Universal Robots URScript: SUB_104.script

def SUB_104():
  global _hidden_verificationVariable=0
  set_target_payload(0.100000, [0.135000, 0.000000, 0.225000], [10.000000, 10.000000, 10.000000, 0.000000, 0.000000, 0.000000])
  set_tool_communication(False, 115200, 0, 1, 1.5, 3.5)
  set_tool_output_mode(0)
  set_tool_digital_output_mode(0, 1)
  set_tool_digital_output_mode(1, 1)
  set_tool_voltage(0)
  set_gravity([0.0, 0.0, 9.82])
  set_tcp(p[0.0,0.06,0.535,0.0,0.0,0.0])
  set_safety_mode_transition_hardness(1)
  set_standard_analog_input_domain(0, 1)
  set_standard_analog_input_domain(1, 1)
  set_tool_analog_input_domain(0, 1)
  set_tool_analog_input_domain(1, 1)
  set_analog_outputdomain(0, 0)
  set_analog_outputdomain(1, 0)
  set_input_actions_to_default()
  set_runstate_gp_boolean_output_to_value(0, 3)
  global isReCapt=False
  global Bucket_Z=[0, 0.7]
  global DistPillar=475
  global CandCnt=0
  global lr=1
  global ReCaptZ=0.05
  global forceval=p[0, 0, 0, 0, 0, 0]
  global CaptDepth=[0.24, 0.48]
  global port=3000
  global isOnlyF=True
  global retX2=p[-0.84412, -0.4876, 0.2794, 0, 0, 1.60139]
  global socket_timeout=120
  global isSkipP=False
  global curpos=p[0, 0, 0, 0, 0, 0]
  global host="192.168.2.2"
  global is_popup=False
  global CaptZOffset=0
  global isGoHome=True
  global i_pos2=p[-0.73382, -0.14132, 0.15275, 1.98953, 2, 0.39506]
  global i_pos1=p[-0.73374, -0.14131, 0.15302, 1.98952, 2.00006, 0.39504]
  global pBucket=[p[0.82565, 0.40576, 0.29486, 0, 0, -1.55844], p[-0.84412, -0.4876, 0.2794, 0, 0, 1.60139]]
  global CaptStepZ=0.08
  global CaptIndex=[0, 0]
  global CaptStepX=0.432
  global pBucketM=p[-0.80141, -0.42542, 0.2879, 0, 0, 1.55713]
  global socket_name="vt"
  global rovi_err=0
  global SubPrgResult=800
  global CurrPos=p[-0.54788, -0.05903, 0.40596, -2.14575, -2.29173, -0.02163]
  global CurrPos_p=p[-0.48377, -0.04896, -0.12847, -2.14575, -2.29173, -0.02163]
  global ForceStartZ=9999
  global Bucket=p[0.32604,0.49174,0.0,-1.882900624652718E-5,2.8304179127934987E-5,-1.593185305749222]
  global BucketM=p[0.32604,0.49174,0.0,1.2814539732933814E-16,-2.611297964559462E-16,-1.5931853071795858]
  global CaptPoint_C=p[-0.4219337985373468,-0.003168602281063755,0.36,-2.1962364319980803,-2.243931608455561,-0.021848848268139726]
  global CaptPoint_C2=p[0.32796661698047924,-0.010768520544682924,0.01931625281283378,2.2288103429550152,-2.213636886217198,8.598462540813273E-5]
  global CaptPoint_L1=p[-0.42193494849366175,-0.2,0.36,-2.1962086037526616,-2.243896582262281,-0.02199725151102503]
  global CaptPoint_L2=p[0.327894307417917,-0.010799940826224014,0.01928712668893995,2.087717047309385,-2.0736781215133306,0.27365839887453103]
  global CaptPoint_R1=p[-0.4219551896101372,0.3,0.36,-2.1960823751566156,-2.243954123514977,-0.021863042557794844]
  global CaptPoint_R2=p[0.327926308680866,-0.010795166414457658,0.019300245403843563,-2.1186306375223185,2.1040550557443427,0.22023197678473694]
  global Capt_1BK_L=p[-0.4574214308482636,-0.48457071473611046,0.3504487959434708,-2.1962343446504526,-2.243967222238911,-0.021809195357489434]
  global Capt_1BK_L_kari=p[-0.9062780457975316,-0.3948152887685301,0.3041579389647211,-1.973454285761923,-1.9354309814821136,0.46582663599327684]
  global Capt_1BK_R=p[-0.4574597285646511,0.4755214243904677,0.35039311859649847,-2.196330286580149,-2.2438949166739053,-0.021738621025254933]
  global Capt_1BK_R_kari=p[-0.9062432457725078,0.5951337546911526,0.30410336812750105,-1.9735777661712788,-1.9353884348839347,0.46584435471052615]
  global Capt_1BK_pos1=p[-0.4218793038724447,-0.003154429464978058,0.2915499891144615,-2.1963422029204875,-2.2438663520270015,-0.02197160668673838]
  global Capt_1BK_pos2=p[-0.42187829024618434,-0.0031710253373066375,0.29156503858953065,-2.196324918349679,-2.2439040699490773,-0.021928444416953782]
  global Capt_1BK_pos2_k=p[-0.6125678682784722,-0.030388805985305904,0.07817890571333086,-1.7892541925095446,-1.8765982468297469,0.6168577595976025]
  global Capt_2BK_L=p[0.42186661528427194,0.4254738068040517,0.35042275762909847,2.239156309475874,-2.1837044610999294,0.002643817066643282]
  global Capt_2BK_L_kari=p[1.0654977997166857,0.48819520122022786,0.0997150581225536,-1.8581624430714432,1.7479280549699192,-0.330138866280949]
  global Capt_2BK_R=p[0.4218208572756906,-0.5427676723257963,0.350372239919558,2.2392697861179327,-2.183553596194912,0.002410470905346486]
  global Capt_2BK_R_kari=p[1.0635189639466671,-0.5406292885234477,0.09156512141204048,-2.1417082668537115,1.7859902718169367,-0.7309097134650204]
  global Capt_2BK_pos1=p[0.42193501458435656,0.004742683868356356,0.35045865974037793,2.2391012408536453,-2.1839704655717003,0.002677867056024068]
  global Capt_2BK_pos2=p[0.421903984494575,0.004707988774967922,0.35045218900915065,2.239114367170047,-2.183895515396197,0.002684056681074047]
  global Capt_2BK_pos2_k=p[0.4977433025854323,-0.009744988529796803,0.07805101846052531,-1.951106747250682,1.9044153054141988,-0.5362260997480872]
  global Capt_GD_M=p[-0.004067001529315755,-0.25244814937804905,-2.093072695775744E-4,0.0332905748643788,-3.1401478399413327,-0.0037841799742876323]
  global Depart_1GD=p[2.9272629556870893E-4,-0.32809839693864495,0.01933497371622539,0.06378642771012696,-3.140731101950783,-3.370184732371461E-4]
  global Depart_LM_2GD=p[-0.022329487227551487,-0.6428077701737687,0.030336146545121845,-0.0656618547018821,2.9888986438241005,0.1566836156643787]
  global Depart_M=p[0.03703236558231149,-0.6428132409158767,-0.02112384231382136,-0.05669816428100925,3.1320592135794345,0.16829522075932857]
  global Depart_RM_2GD=p[0.10304778501057178,-0.6389514408512296,0.030085893950939302,0.039485966396909634,-3.0126453050861945,-0.17126767917269797]
  global Depsrt_2GD=p[3.027477292580124E-4,-0.3281073069657892,0.019292078494201337,0.06380062875024692,-3.1406974312388685,-3.876005598966342E-4]
  global HomePointL=p[-0.36789,-0.5117344641471838,0.78,-0.6278857271586024,3.0680899128661667,-8.649957362498864E-4]
  global PickPos=p[0.10830682331105715,-1.3709505888096256,-0.18404188875951455,-0.00622194000158997,2.880236948927292,-0.00383636509397631]
  global Solve=p[-0.00368,-0.0021000000000000003,0.25739999999999996,0.0,0.0,0.0]
  global TEST=p[0.1,0.0,0.2,0.0,0.0,0.0]
  global UF=p[0.0,0.0,0.0,0.0,0.0,0.0]
  global g1CV_1_M=p[0.29093319989156785,-0.9405344885124904,-0.08686754932079166,1.9884186265311852,2.2323374792844253,0.1524643645929425]
  global g1CV_posL1=p[0.05028133628211688,-0.4526481033729615,0.1221845548632916,-2.213335080948508,-2.1937561336067057,-0.3280056759040735]
  global g1CV_posR1=p[0.03743870476062511,-0.53119407812668,0.11301901343688614,2.073418671558482,2.153257467049566,0.11656306439039889]
  global g1GD_pos1=p[0.06841781024889843,-0.5456037307108855,0.367146167315866,2.4108578981103275,1.7957834606331096,0.12544942012730473]
  global g1GD_pos2=p[-0.38705506163240566,-0.3905161646272917,0.3670805000411974,2.9334800678601534,0.5562338866571123,0.025147235284150155]
  global g1GD_pos3=p[-0.614523200343285,-0.009392732880809615,0.3783325239377683,2.0687271625579515,2.17319336139756,0.21682066343437634]
  global g1GD_pos4=p[-0.4351564513137486,0.028155221259926276,0.13086718327275837,2.2072871432536783,2.2307343865376095,-0.0018307218179379997]
  global g1GD_pos5=p[-0.8151645021025727,-0.01706756320728201,0.08179601375099321,2.212895896456039,2.218350348620789,0.019350113017735118]
  global g1GD_posL1=p[-0.08276848269606216,-0.3996147100031649,0.1488453551331823,2.286527078917204,1.8420745504477611,0.33698451773695576]
  global g1GD_posL2=p[-0.3253977027403738,-0.3024804624281039,0.16332814085945146,2.72312820760317,0.9631021078169197,0.32447452035226126]
  global g1GD_posL3=p[-0.6791033397183219,0.06787475590683856,0.16337212788108813,2.1383125299263996,2.086116032377724,0.4536080263755059]
  global g1GD_posR1=p[-0.09893370538053747,-0.4999608954567234,0.14329885217724153,2.43311852414254,1.4238397520832589,0.08559216753941556]
  global g1GD_posR2=p[-0.3729565201882258,-0.3752983669473301,0.143299052800563,2.6951655216297596,0.8130506811102118,-0.02387549506099888]
  global g1GD_posR3=p[-0.7385929502572233,-0.029472684480355026,0.1499650660949685,2.0484522752014467,1.9493695704119496,0.18368227556562683]
  global g2CV_1_M=p[0.2880593256931911,-0.933809998732841,-0.08698643380656113,2.0727630257838867,2.230596497566155,0.15036691287620893]
  global g2CV_posL1=p[0.3409386496330911,-0.4656338066361442,0.1250074988128972,2.209372209162659,2.1945371304665926,0.3160714960040194]
  global g2CV_posR1=p[0.3400736278759575,-0.531334269888987,0.1183415684753657,2.07314649492589,2.1532617466521136,0.11638666128062146]
  global g2GD_pos1=p[0.3390086633742754,-0.5203839341398588,0.22258,2.022696172282159,2.259224887850344,0.09811005079237367]
  global g2GD_pos2=p[0.4140891885236144,0.14850105084950693,0.1582916370575993,-0.10302503203970696,3.1008909166713883,0.18748967846962497]
  global g2GD_pos3=p[0.32377086541216454,-0.01023215987367155,0.15821240334102793,2.279746475463588,-2.06129961332614,-0.16578334012307952]
  global g2GD_pos4=p[0.7398823109797592,-0.026643494293930835,0.22255839224074236,2.162283599874437,-2.168919538925757,-0.13861635932587069]
  global g2GD_pos5=p[0.22271243238356278,-0.026679271241024524,0.22257782526136982,1.3056143664331146,-2.8077458860488136,-0.17177240522535248]
  global gCV_11_M=p[0.3028468774759881,-0.9375366886748661,-0.09782511939875749,1.9971971468330036,2.0934336167121885,0.3604928446251781]
  global gCV_12_M=p[0.34776610649632045,-0.9364202289953052,-0.09784932758070936,1.9972781240484352,2.0934384510830295,0.3604701319279358]
  global gCV_13_M=p[0.43083047728791135,-0.9363258116427577,0.028711300566433673,1.9972504931093251,2.0935710325846095,0.3605630596092243]
  global gCV_14=p[0.35645641620611146,-0.8914305774826713,-0.17737239800677018,2.1506886654737776,2.1461343800624295,0.40986447399780934]
  global gCV_15=p[0.4370373250739419,-0.891408661166693,-0.1773997714481486,2.1507483614991094,2.1461657601704176,0.40983132876462236]
  global gCV_16=p[0.4597123429384979,-0.8913837618729653,-0.03599504377258328,2.1506156333226136,2.1462305295546718,0.4099109158136618]
  global gCV_17=p[0.037528034463104695,-0.6904892259828748,-0.12243237639232962,-0.12012393052395552,2.832430475095037,0.48967048060305135]
  global gCV_18=p[0.03600103065313248,-0.6368623043127666,-0.12241687036449483,-0.12010351348807546,2.832474314609516,0.48970816626953567]
  global gCV_2_M=p[0.2909259851094176,-0.9405632657218349,0.07217586581493451,1.9883998690824036,2.232303337331875,0.15240099649164607]
  global gCV_3_M=p[0.29099390607376485,-0.6570558385379063,0.0722153583041818,1.9884242634571576,2.2321538498123994,0.15249643504377583]
  global gCV_5=p[0.045776199142861046,-0.9791473230816141,0.8415069045351792,2.0229894037377316,2.080009888728606,0.35618099403901887]
  global gCV_pos5=p[0.3400172856834047,-0.9722754606605235,-0.18287928563575456,2.073394561413637,2.1531827558666565,0.11639000988241816]
  global gGD_100_1LM=p[0.04146780808756359,-0.6870904124925177,-0.1232943093634104,-0.006305250057386166,-2.863965809273829,-0.5082528300185785]
  global gGD_1_LM=p[0.03230475520524248,-0.7130493639313011,-0.12313048496237139,-0.146861070648958,2.82789794799972,0.5264874367071143]
  global gGD_1_M=p[0.03530347986661216,-0.7127417041043018,-0.12310155616185803,-0.05957601747684272,3.087266550524023,0.5413331493142363]
  global gGD_1_MM=p[0.03527332731929103,-0.7200324399236822,-0.12309145975746483,-0.05946537723025455,3.087281488106925,0.5412792107775745]
  global gGD_1_RM=p[0.03790072787181614,-0.7120178370098972,-0.12342664631367783,0.016248473772828512,-2.8629005997783534,-0.4984191911686871]
  global gGD_200_2LM=p[0.04175812558137225,-0.6358261219893102,-0.12285474020423298,-0.006257718193554584,-2.863964784148567,-0.5084621939645108]
  global gGD_2_LM=p[0.030572718129261614,-0.6604571464977577,-0.12310155388330796,-0.14682775034190318,2.827796436074414,0.5264394416290918]
  global gGD_2_M=p[0.03435287261256309,-0.6587000226205477,-0.12439339172019714,-0.05966040009453588,3.0872872080206544,0.5411228747416044]
  global gGD_2_RM=p[0.036719806244467246,-0.6603323308238997,-0.12407566124392316,0.01621270878011713,-2.862858880050919,-0.4984088290677938]
  global gGD_300_3LM=p[0.04182050265947469,-0.6066076810742604,-0.03602288107395374,-0.006290924000441408,-2.8640915241774816,-0.5083501301248439]
  global gGD_3_LM=p[0.03053842874056699,-0.6329626532416066,-0.03639755844951337,-0.14684511442606807,2.8278657439893307,0.5264948582193963]
  global gGD_3_M=p[0.03430957843779042,-0.6330568980917707,-0.04259950182125549,-0.05969688861307265,3.087293602983763,0.5413247841490268]
  global gGD_3_RM=p[0.03673432946585267,-0.632032638942058,-0.03445023119106272,0.016317873028914045,-2.8628788700289953,-0.4985371510851901]
  global gGD_400_1RM=p[0.03765496539143813,-0.6905733748742057,-0.12240702670509729,-0.12009639012349203,2.8324503628258273,0.48945657912051843]
  global gGD_4_LM=p[-0.050697518013391604,-0.4788149830819543,0.04525080740157289,-0.14673385744666134,2.827848291285266,0.5267055795817903]
  global gGD_4_RM=p[0.10921584432919978,-0.48073334437858256,0.06990685637741062,0.016338390530391603,-2.862804566994448,-0.49861203356258266]
  global gGD_500_2RM=p[0.0364038044475721,-0.6361408639594927,-0.1228896102948493,-0.12001814478849077,2.8324363686538967,0.4895422385690364]
  global gGD_600_3RM=p[0.03597788557419286,-0.6039591135870097,-0.03251312847845622,-0.12016380804709932,2.832584395249392,0.4895204315491753]
  global gGD_M_20=p[0.03524102305764369,-0.704963855446233,-0.12310321086399345,-0.05961230604660993,3.0873078767639504,0.5414261100507907]
  global gGD_M_30=p[0.03527181411394771,-0.6949613298581867,-0.12309199448652725,-0.05962447301074729,3.087287038166274,0.5412100180254447]
  global gGD_M_40=p[0.035236425258241534,-0.6834410208824955,-0.12309554834290798,-0.05953064339288712,3.087315110349415,0.5412921265180426]
  global gHome_Position=p[3.053061697190075E-4,-0.3281132156787397,0.01930332806480972,0.0637196994340987,-3.140722020313799,-3.2847660283345163E-4]
  step_count_d97aa564_60a0_4340_971f_70619f182064 = 0.0
  thread Step_Counter_Thread_19d9c95c_4707_4bf0_be0f_94ec4e598e3f():
    while (True):
      step_count_d97aa564_60a0_4340_971f_70619f182064 = step_count_d97aa564_60a0_4340_971f_70619f182064 + 1.0
      sync()
    end
  end
  run Step_Counter_Thread_19d9c95c_4707_4bf0_be0f_94ec4e598e3f()
  global tm_200=0
  global tm_200_is_counting=False
  thread Timer_Thread():
    while (True):
      if (tm_200_is_counting):
        tm_200 = tm_200 + get_steptime()
      end
      sync()
    end
  end
  run Timer_Thread()
  while (True):
    $ 2 "ロボットプログラム"
    $ 3 "SET_BUCKET()"
    SET_BUCKET()
    $ 4 "ROVI_CAPTURE"
    $ 6 "If文 ( not ROVI_CAPTURE())"
    if ((  not  ROVI_CAPTURE())):
      $ 7 "SubPrgResult:=rovi_err"
      global SubPrgResult=rovi_err
      $ 8 "待機: 999999.0"
      sleep(999999.0)
    end
    $ 10 "If文 (CandCnt<1)"
    if ((CandCnt<1)):
      $ 11 "SubPrgResult:=990"
      global SubPrgResult=990
      $ 12 "待機: 999999.0"
      sleep(999999.0)
    end
    $ 13 "ROVI_SOLVE"
    $ 14 "If文 (CandCnt>0)"
    if ((CandCnt>0)):
      $ 16 "retX2:=ROVI_SOLVE()"
      global retX2=ROVI_SOLVE()
      $ 18 "If文 (retX2[0]≟10000.)"
      if ((retX2[0] == 10000.)):
        $ 19 "SubPrgResult:=rovi_err"
        global SubPrgResult=rovi_err
        $ 20 "待機: 999999.0"
        sleep(999999.0)
      end
    end
    $ 23 "UF:=retX2"
    global UF=retX2
    $ 24 "If文 (is_popup)"
    if ((is_popup)):
      $ 25 "ポップアップ: ROVI_SOLVE succeed."
      popup("ROVI_SOLVE succeed.", "メッセージ", False, False, blocking=True)
    end
    $ 26 "PICK"
    $ 27 "荷重の設定: k10"
    set_target_payload(0.100000, [0.135000, 0.000000, 0.225000], [10.000000, 10.000000, 10.000000, 0.000000, 0.000000, 0.000000])
    $ 28 "pillar:=CHECK_PILLAR()"
    global pillar=CHECK_PILLAR()
    $ 29 "If文 (GPBI_WorkExists≠ True )"
    global thread_flag_29=0
    thread Thread_if_29():
      $ 30 "If文 (pillar≟1)"
      if ((pillar == 1)):
        $ 32 "MoveL"
        $ 33 "gGD_4_LM" "breakAfter"
        set_tcp(p[0.0,0.06,0.535,0.0,0.0,0.0])
        movel(pose_trans(UF, gGD_4_LM), a=0.14, v=0.4)
        $ 34 "gGD_3_LM" "breakAfter"
        set_tcp(p[0.0,0.06,0.535,0.0,0.0,0.0])
        movel(pose_trans(UF, gGD_3_LM), a=0.14, v=0.4)
        $ 35 "gGD_2_LM" "breakAfter"
        set_tcp(p[0.0,0.06,0.535,0.0,0.0,0.0])
        movel(pose_trans(UF, gGD_2_LM), a=0.14, v=0.4)
        $ 37 "待機: 0.5"
        sleep(0.5)
        $ 38 "gGD_1_LM" "breakAfter"
        set_tcp(p[0.0,0.06,0.535,0.0,0.0,0.0])
        movel(pose_trans(UF, gGD_1_LM), a=0.14, v=0.4)
      else:
        $ 39 "ElseIf (pillar≟2)"
        if ((pillar == 2)):
          $ 41 "MoveL"
          $ 42 "gGD_4_RM" "breakAfter"
          set_tcp(p[0.0,0.06,0.535,0.0,0.0,0.0])
          movel(pose_trans(UF, gGD_4_RM), a=0.14, v=0.4)
          $ 43 "gGD_3_RM" "breakAfter"
          set_tcp(p[0.0,0.06,0.535,0.0,0.0,0.0])
          movel(pose_trans(UF, gGD_3_RM), a=0.14, v=0.4)
          $ 44 "gGD_2_RM" "breakAfter"
          set_tcp(p[0.0,0.06,0.535,0.0,0.0,0.0])
          movel(pose_trans(UF, gGD_2_RM), a=0.14, v=0.4)
          $ 46 "待機: 0.5"
          sleep(0.5)
          $ 47 "gGD_1_RM" "breakAfter"
          set_tcp(p[0.0,0.06,0.535,0.0,0.0,0.0])
          movel(pose_trans(UF, gGD_1_RM), a=0.14, v=0.4)
        else:
          $ 48 "Else" "noBreak"
          $ 49 "If文 (DistPillar≥0)"
          if ((DistPillar >= 0)):
            $ 50 "If文 (is_popup)"
            if ((is_popup)):
              $ 51 "ポップアップ: center L"
              popup("center L", "メッセージ", False, False, blocking=True)
            end
            $ 52 "MoveL"
            $ 53 "gGD_3_M" "breakAfter"
            set_tcp(p[0.0,0.06,0.535,0.0,0.0,0.0])
            movel(pose_trans(UF, gGD_3_M), a=0.14, v=0.4)
            $ 54 "gGD_2_M" "breakAfter"
            set_tcp(p[0.0,0.06,0.535,0.0,0.0,0.0])
            movel(pose_trans(UF, gGD_2_M), a=0.14, v=0.4)
            $ 55 "tm_200: 停止"
            tm_200_is_counting = False
            $ 56 "i_pos1:=get_actual_tcp_pose()"
            global i_pos1= get_actual_tcp_pose ()
            $ 57 "i_pos2:=get_target_tcp_pose()"
            global i_pos2= get_target_tcp_pose ()
            $ 58 "If文 (is_popup)"
            if ((is_popup)):
              $ 59 "ポップアップ: clamp ready"
              popup("clamp ready", "メッセージ", False, False, blocking=True)
            end
            $ 61 "待機: 0.5"
            sleep(0.5)
            $ 62 "gGD_M_30" "breakAfter"
            set_tcp(p[0.0,0.06,0.535,0.0,0.0,0.0])
            movel(pose_trans(UF, gGD_M_30), a=0.14, v=0.4)
          else:
            $ 64 "Else" "noBreak"
            $ 66 "MoveL"
            $ 67 "gGD_3_M" "breakAfter"
            set_tcp(p[0.0,0.06,0.535,0.0,0.0,0.0])
            movel(pose_trans(UF, gGD_3_M), a=0.14, v=0.5)
            $ 68 "gGD_2_M" "breakAfter"
            set_tcp(p[0.0,0.06,0.535,0.0,0.0,0.0])
            movel(pose_trans(UF, gGD_2_M), a=0.14, v=0.5)
            $ 69 "i_pos1:=get_actual_tcp_pose()"
            global i_pos1= get_actual_tcp_pose ()
            $ 70 "i_pos2:=get_target_tcp_pose()"
            global i_pos2= get_target_tcp_pose ()
            $ 72 "待機: 0.5"
            sleep(0.5)
            $ 73 "gGD_M_30" "breakAfter"
            set_tcp(p[0.0,0.06,0.535,0.0,0.0,0.0])
            movel(pose_trans(UF, gGD_M_30), a=0.14, v=0.5)
          end
        end
      end
      thread_flag_29 = 1
    end
    if ((read_input_boolean_register(9) !=   True  )):
      global thread_handler_29=run Thread_if_29()
      while (thread_flag_29 == 0):
        if not((read_input_boolean_register(9) !=   True  )):
          kill thread_handler_29
          thread_flag_29 = 2
        else:
          sync()
        end
      end
    else:
      thread_flag_29 = 2
    end
    $ 76 "If文 (is_popup)"
    if ((is_popup)):
      $ 77 "ポップアップ: Clamp OK?"
      popup("Clamp OK?", "メッセージ", False, False, blocking=True)
    end
  end
end
